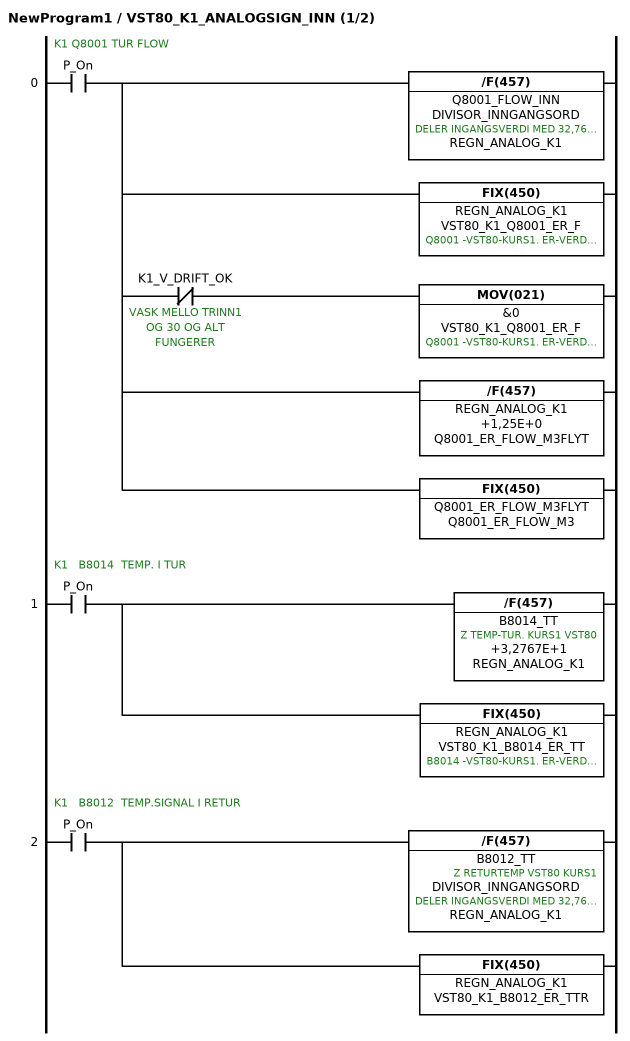
; [picture p144: NewProgram1 / VST80_K1_ANALOGSIGN_INN, rungs 0-2]
; rung 0: K1 Q8001 TUR FLOW
LD P_On
OUT TR0
/F(457) Q8001_FLOW_INN DIVISOR_INNGANGSORD REGN_ANALOG_K1  ; DELER INGANGSVERDI MED 32,760 FOR OMREGNING TIL 0-1000
FIX(450) REGN_ANALOG_K1 VST80_K1_Q8001_ER_F  ; Q8001 -VST80-KURS1. ER-VERDI FLOW I TUR
ANDNOT K1_V_DRIFT_OK  ; VASK MELLO TRINN1 OG 30 OG ALT FUNGERER
MOV(021) &0 VST80_K1_Q8001_ER_F  ; Q8001 -VST80-KURS1. ER-VERDI FLOW I TUR
LD TR0
/F(457) REGN_ANALOG_K1 +1,25E+0 Q8001_ER_FLOW_M3FLYT
FIX(450) Q8001_ER_FLOW_M3FLYT Q8001_ER_FLOW_M3
; rung 1: K1   B8014  TEMP. I TUR
LD P_On
/F(457) B8014_TT +3,2767E+1 REGN_ANALOG_K1  ; Z TEMP-TUR. KURS1 VST80
FIX(450) REGN_ANALOG_K1 VST80_K1_B8014_ER_TT  ; B8014 -VST80-KURS1. ER-VERDI TEMPERATUR I TUR TIL VST
; rung 2: K1   B8012  TEMP.SIGNAL I RETUR
LD P_On
/F(457) B8012_TT DIVISOR_INNGANGSORD REGN_ANALOG_K1  ; Z RETURTEMP VST80 KURS1, DELER INGANGSVERDI MED 32,760 FOR OMREGNING TIL 0-1000
FIX(450) REGN_ANALOG_K1 VST80_K1_B8012_ER_TTR

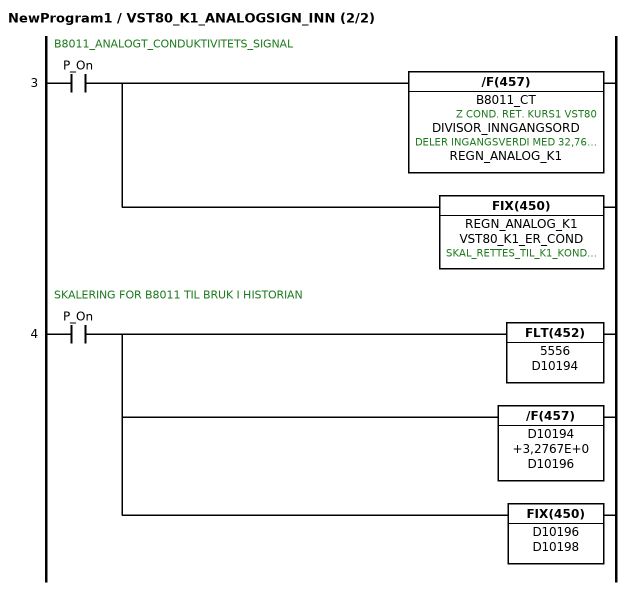
; rung 3: B8011_ANALOGT_CONDUKTIVITETS_SIGNAL
LD P_On
/F(457) B8011_CT DIVISOR_INNGANGSORD REGN_ANALOG_K1  ; Z COND. RET. KURS1 VST80, DELER INGANGSVERDI MED 32,760 FOR OMREGNING TIL 0-1000
FIX(450) REGN_ANALOG_K1 VST80_K1_ER_COND  ; SKAL_RETTES_TIL_K1_KOND_ERVERDI
; rung 4: SKALERING FOR B8011 TIL BRUK I HISTORIAN
LD P_On
FLT(452) 5556 D10194
/F(457) D10194 +3,2767E+0 D10196
FIX(450) D10196 D10198

### Section VST80_K1_GRAF_FEIL_TXT

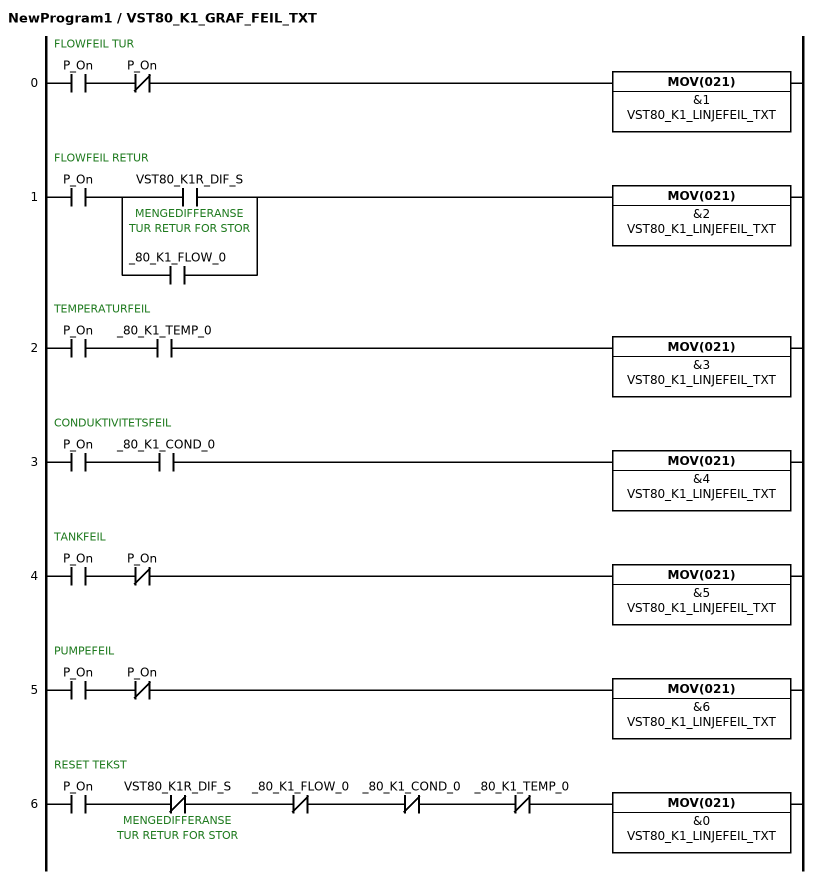
; rung 0: FLOWFEIL TUR
LD P_On
ANDNOT P_On
MOV(021) &1 VST80_K1_LINJEFEIL_TXT
; rung 1: FLOWFEIL RETUR
LD P_On
LD VST80_K1R_DIF_S  ; MENGEDIFFERANSE TUR RETUR FOR STOR
OR _80_K1_FLOW_0
ANDLD
MOV(021) &2 VST80_K1_LINJEFEIL_TXT
; rung 2: TEMPERATURFEIL
LD P_On
AND _80_K1_TEMP_0
MOV(021) &3 VST80_K1_LINJEFEIL_TXT
; rung 3: CONDUKTIVITETSFEIL
LD P_On
AND _80_K1_COND_0
MOV(021) &4 VST80_K1_LINJEFEIL_TXT
; rung 4: TANKFEIL
LD P_On
ANDNOT P_On
MOV(021) &5 VST80_K1_LINJEFEIL_TXT
; rung 5: PUMPEFEIL
LD P_On
ANDNOT P_On
MOV(021) &6 VST80_K1_LINJEFEIL_TXT
; rung 6: RESET TEKST
LD P_On
ANDNOT VST80_K1R_DIF_S  ; MENGEDIFFERANSE TUR RETUR FOR STOR
ANDNOT _80_K1_FLOW_0
ANDNOT _80_K1_COND_0
ANDNOT _80_K1_TEMP_0
MOV(021) &0 VST80_K1_LINJEFEIL_TXT

### Section VST80_K1_MENGDE_FASESKIFT

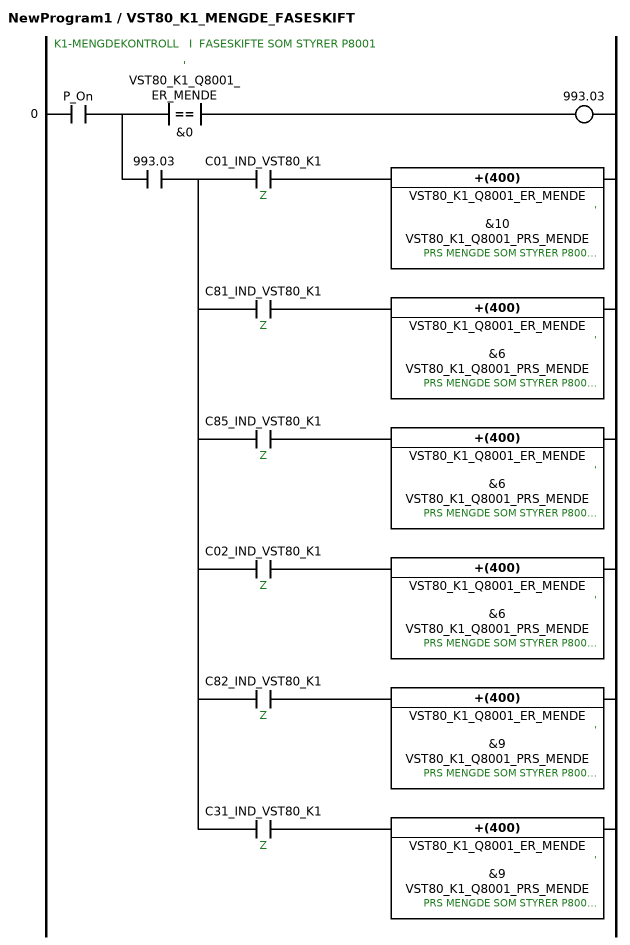
; rung 0: K1-MENGDEKONTROLL   I  FASESKIFTE SOM STYRER P8001
LD P_On
OUT TR0
AND=(300) VST80_K1_Q8001_ER_MENDE &0  ; '
OUT 993.03
LD TR0
AND 993.03
OUT TR0
AND C01_IND_VST80_K1  ; Z
+(400) VST80_K1_Q8001_ER_MENDE &10 VST80_K1_Q8001_PRS_MENDE  ; ', PRS MENGDE SOM STYRER P8001 VED FASESKIFTE
LD TR0
AND C81_IND_VST80_K1  ; Z
+(400) VST80_K1_Q8001_ER_MENDE &6 VST80_K1_Q8001_PRS_MENDE  ; ', PRS MENGDE SOM STYRER P8001 VED FASESKIFTE
LD TR0
AND C85_IND_VST80_K1  ; Z
+(400) VST80_K1_Q8001_ER_MENDE &6 VST80_K1_Q8001_PRS_MENDE  ; ', PRS MENGDE SOM STYRER P8001 VED FASESKIFTE
LD TR0
AND C02_IND_VST80_K1  ; Z
+(400) VST80_K1_Q8001_ER_MENDE &6 VST80_K1_Q8001_PRS_MENDE  ; ', PRS MENGDE SOM STYRER P8001 VED FASESKIFTE
LD TR0
AND C82_IND_VST80_K1  ; Z
+(400) VST80_K1_Q8001_ER_MENDE &9 VST80_K1_Q8001_PRS_MENDE  ; ', PRS MENGDE SOM STYRER P8001 VED FASESKIFTE
LD TR0
AND C31_IND_VST80_K1  ; Z
+(400) VST80_K1_Q8001_ER_MENDE &9 VST80_K1_Q8001_PRS_MENDE  ; ', PRS MENGDE SOM STYRER P8001 VED FASESKIFTE

### Section VST80_K1_TR_VEKS
; VST80 KURS1 VEKSLING AV TRINN.

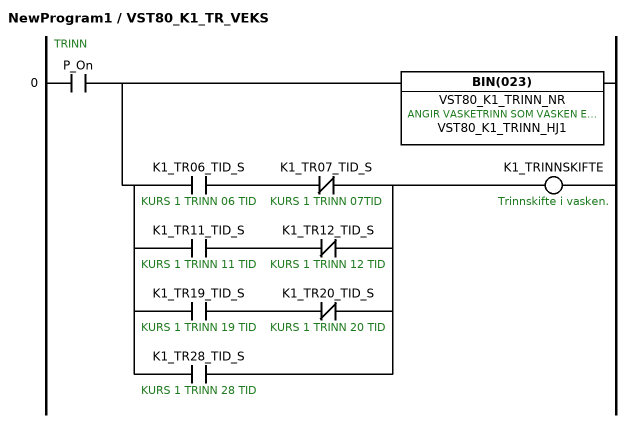
; rung 0: TRINN
LD P_On
BIN(023) VST80_K1_TRINN_NR VST80_K1_TRINN_HJ1  ; ANGIR VASKETRINN SOM VASKEN ER I
LD K1_TR06_TID_S  ; KURS 1 TRINN 06 TID
ANDNOT K1_TR07_TID_S  ; KURS 1 TRINN 07TID
LD K1_TR11_TID_S  ; KURS 1 TRINN 11 TID
ANDNOT K1_TR12_TID_S  ; KURS 1 TRINN 12 TID
ORLD
LD K1_TR19_TID_S  ; KURS 1 TRINN 19 TID
ANDNOT K1_TR20_TID_S  ; KURS 1 TRINN 20 TID
ORLD
OR K1_TR28_TID_S  ; KURS 1 TRINN 28 TID
ANDLD
OUT K1_TRINNSKIFTE  ; Trinnskifte i vasken.

### Section VST80_K1_FEIL_RET
; FEIL I RETUR / FLOW / TEMP / COND

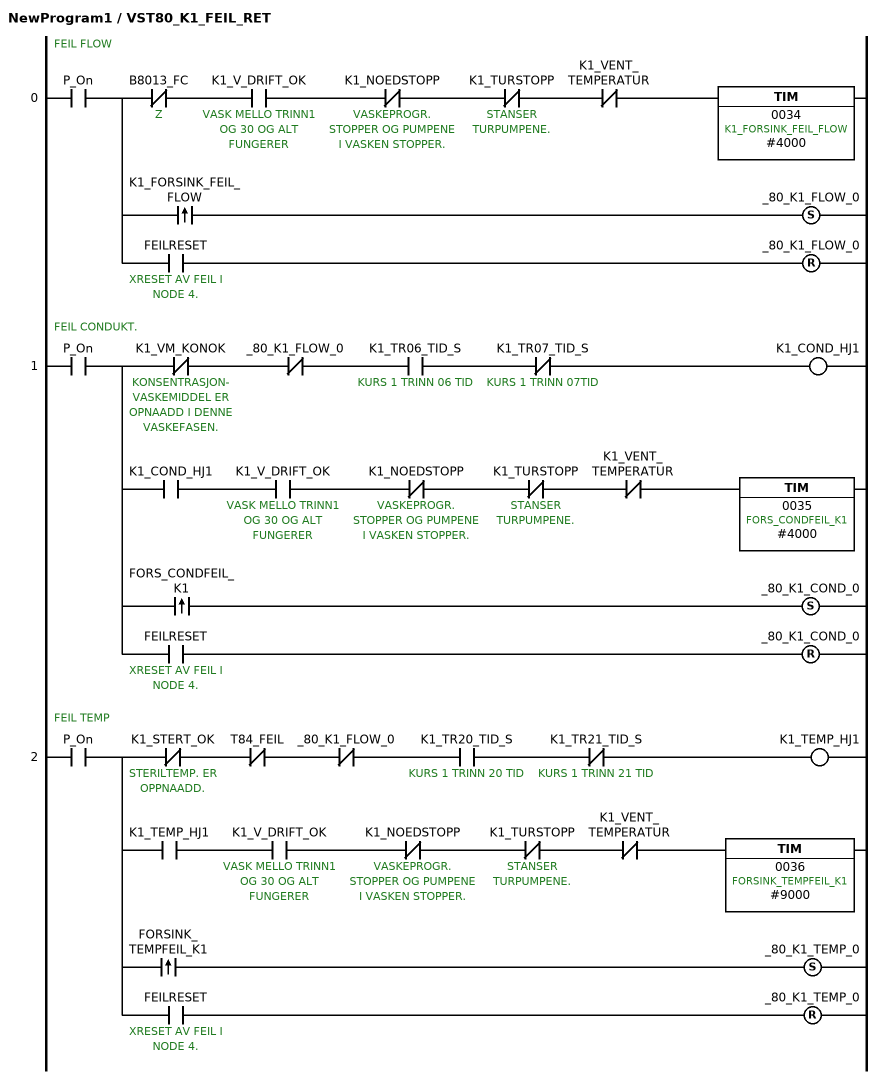
; rung 0: FEIL FLOW
LD P_On
OUT TR0
ANDNOT B8013_FC  ; Z
AND K1_V_DRIFT_OK  ; VASK MELLO TRINN1 OG 30 OG ALT FUNGERER
ANDNOT K1_NOEDSTOPP  ; VASKEPROGR. STOPPER OG PUMPENE I VASKEN STOPPER.
ANDNOT K1_TURSTOPP  ; STANSER TURPUMPENE.
ANDNOT K1_VENT_TEMPERATUR
TIM 0034 #4000  ; K1_FORSINK_FEIL_FLOW
LD TR0
@AND K1_FORSINK_FEIL_FLOW
SET _80_K1_FLOW_0
LD TR0
AND FEILRESET  ; XRESET AV FEIL I NODE 4.
RSET _80_K1_FLOW_0
; rung 1: FEIL CONDUKT.
LD P_On
OUT TR0
ANDNOT K1_VM_KONOK  ; KONSENTRASJON-VASKEMIDDEL ER OPNAADD I DENNE VASKEFASEN.
ANDNOT _80_K1_FLOW_0
AND K1_TR06_TID_S  ; KURS 1 TRINN 06 TID
ANDNOT K1_TR07_TID_S  ; KURS 1 TRINN 07TID
OUT K1_COND_HJ1
LD TR0
AND K1_COND_HJ1
AND K1_V_DRIFT_OK  ; VASK MELLO TRINN1 OG 30 OG ALT FUNGERER
ANDNOT K1_NOEDSTOPP  ; VASKEPROGR. STOPPER OG PUMPENE I VASKEN STOPPER.
ANDNOT K1_TURSTOPP  ; STANSER TURPUMPENE.
ANDNOT K1_VENT_TEMPERATUR
TIM 0035 #4000  ; FORS_CONDFEIL_K1
LD TR0
@AND FORS_CONDFEIL_K1
SET _80_K1_COND_0
LD TR0
AND FEILRESET  ; XRESET AV FEIL I NODE 4.
RSET _80_K1_COND_0
; rung 2: FEIL TEMP
LD P_On
OUT TR0
ANDNOT K1_STERT_OK  ; STERILTEMP. ER OPPNAADD.
ANDNOT T84_FEIL
ANDNOT _80_K1_FLOW_0
AND K1_TR20_TID_S  ; KURS 1 TRINN 20 TID
ANDNOT K1_TR21_TID_S  ; KURS 1 TRINN 21 TID
OUT K1_TEMP_HJ1
LD TR0
AND K1_TEMP_HJ1
AND K1_V_DRIFT_OK  ; VASK MELLO TRINN1 OG 30 OG ALT FUNGERER
ANDNOT K1_NOEDSTOPP  ; VASKEPROGR. STOPPER OG PUMPENE I VASKEN STOPPER.
ANDNOT K1_TURSTOPP  ; STANSER TURPUMPENE.
ANDNOT K1_VENT_TEMPERATUR
TIM 0036 #9000  ; FORSINK_TEMPFEIL_K1
LD TR0
@AND FORSINK_TEMPFEIL_K1
SET _80_K1_TEMP_0
LD TR0
AND FEILRESET  ; XRESET AV FEIL I NODE 4.
RSET _80_K1_TEMP_0

### Section VST80_K1_VASKERAPPORT
; VST80 / KURS1 VASKERAPPORT

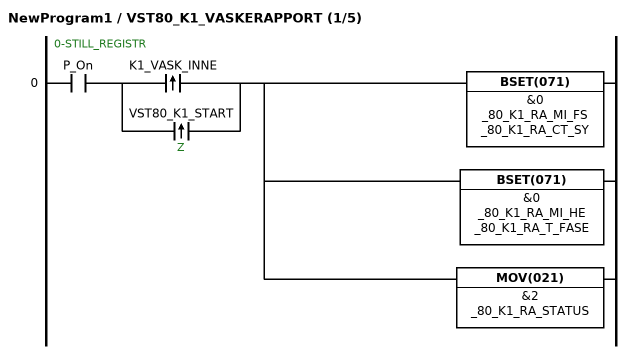
; rung 0: 0-STILL_REGISTR
LD P_On
@LD K1_VASK_INNE
@OR VST80_K1_START  ; Z
ANDLD
BSET(071) &0 _80_K1_RA_MI_FS _80_K1_RA_CT_SY
BSET(071) &0 _80_K1_RA_MI_HE _80_K1_RA_T_FASE
MOV(021) &2 _80_K1_RA_STATUS

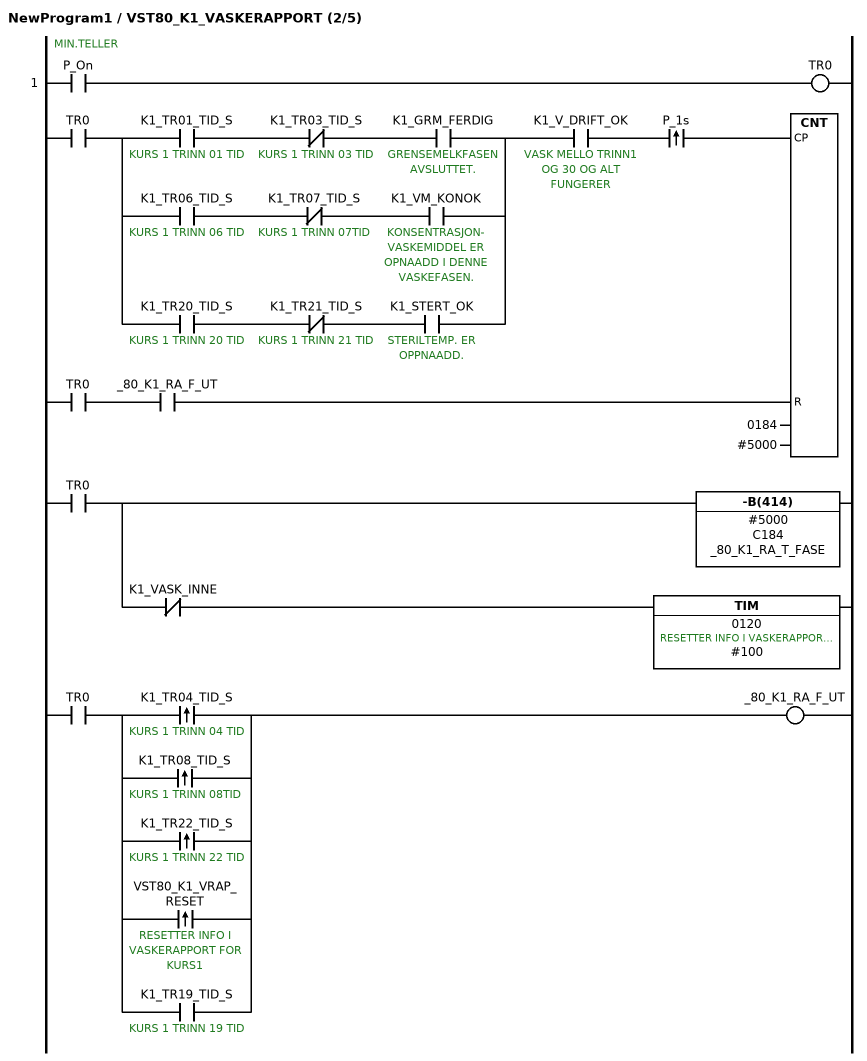
; rung 1: MIN.TELLER
LD P_On
OUT TR0
LD K1_TR01_TID_S  ; KURS 1 TRINN 01 TID
ANDNOT K1_TR03_TID_S  ; KURS 1 TRINN 03 TID
AND K1_GRM_FERDIG  ; GRENSEMELKFASEN AVSLUTTET.
LD K1_TR06_TID_S  ; KURS 1 TRINN 06 TID
ANDNOT K1_TR07_TID_S  ; KURS 1 TRINN 07TID
AND K1_VM_KONOK  ; KONSENTRASJON-VASKEMIDDEL ER OPNAADD I DENNE VASKEFASEN.
ORLD
LD K1_TR20_TID_S  ; KURS 1 TRINN 20 TID
ANDNOT K1_TR21_TID_S  ; KURS 1 TRINN 21 TID
AND K1_STERT_OK  ; STERILTEMP. ER OPPNAADD.
ORLD
ANDLD
AND K1_V_DRIFT_OK  ; VASK MELLO TRINN1 OG 30 OG ALT FUNGERER
@AND P_1s
LD TR0
AND _80_K1_RA_F_UT
CNT 0184 #5000
LD TR0
-B(414) #5000 C184 _80_K1_RA_T_FASE
ANDNOT K1_VASK_INNE
TIM 0120 #100  ; RESETTER INFO I VASKERAPPORT FOR KURS1
LD TR0
@LD K1_TR04_TID_S  ; KURS 1 TRINN 04 TID
@OR K1_TR08_TID_S  ; KURS 1 TRINN 08TID
@OR K1_TR22_TID_S  ; KURS 1 TRINN 22 TID
@OR VST80_K1_VRAP_RESET  ; RESETTER INFO I VASKERAPPORT FOR KURS1
OR K1_TR19_TID_S  ; KURS 1 TRINN 19 TID
ANDLD
OUT _80_K1_RA_F_UT

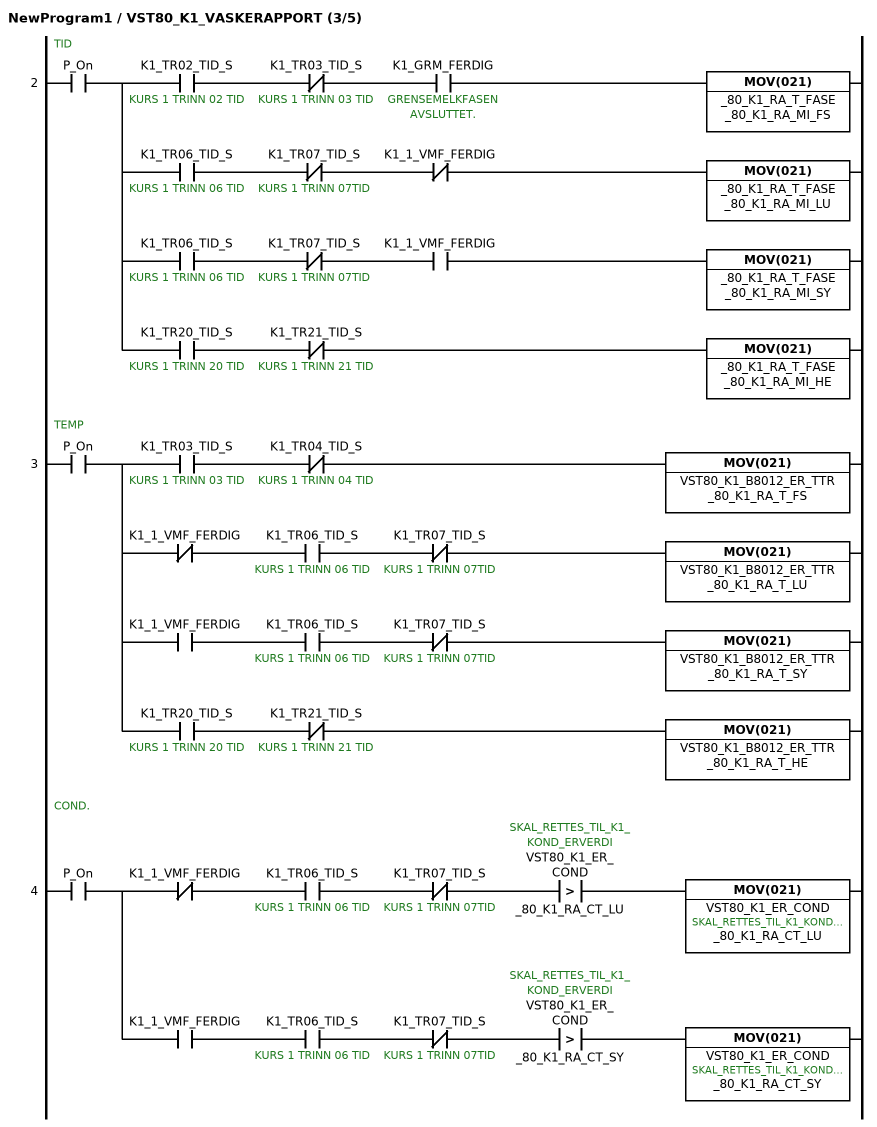
; rung 2: TID
LD P_On
OUT TR0
AND K1_TR02_TID_S  ; KURS 1 TRINN 02 TID
ANDNOT K1_TR03_TID_S  ; KURS 1 TRINN 03 TID
AND K1_GRM_FERDIG  ; GRENSEMELKFASEN AVSLUTTET.
MOV(021) _80_K1_RA_T_FASE _80_K1_RA_MI_FS
LD TR0
AND K1_TR06_TID_S  ; KURS 1 TRINN 06 TID
ANDNOT K1_TR07_TID_S  ; KURS 1 TRINN 07TID
ANDNOT K1_1_VMF_FERDIG
MOV(021) _80_K1_RA_T_FASE _80_K1_RA_MI_LU
LD TR0
AND K1_TR06_TID_S  ; KURS 1 TRINN 06 TID
ANDNOT K1_TR07_TID_S  ; KURS 1 TRINN 07TID
AND K1_1_VMF_FERDIG
MOV(021) _80_K1_RA_T_FASE _80_K1_RA_MI_SY
LD TR0
AND K1_TR20_TID_S  ; KURS 1 TRINN 20 TID
ANDNOT K1_TR21_TID_S  ; KURS 1 TRINN 21 TID
MOV(021) _80_K1_RA_T_FASE _80_K1_RA_MI_HE
; rung 3: TEMP
LD P_On
OUT TR0
AND K1_TR03_TID_S  ; KURS 1 TRINN 03 TID
ANDNOT K1_TR04_TID_S  ; KURS 1 TRINN 04 TID
MOV(021) VST80_K1_B8012_ER_TTR _80_K1_RA_T_FS
LD TR0
ANDNOT K1_1_VMF_FERDIG
AND K1_TR06_TID_S  ; KURS 1 TRINN 06 TID
ANDNOT K1_TR07_TID_S  ; KURS 1 TRINN 07TID
MOV(021) VST80_K1_B8012_ER_TTR _80_K1_RA_T_LU
LD TR0
AND K1_1_VMF_FERDIG
AND K1_TR06_TID_S  ; KURS 1 TRINN 06 TID
ANDNOT K1_TR07_TID_S  ; KURS 1 TRINN 07TID
MOV(021) VST80_K1_B8012_ER_TTR _80_K1_RA_T_SY
LD TR0
AND K1_TR20_TID_S  ; KURS 1 TRINN 20 TID
ANDNOT K1_TR21_TID_S  ; KURS 1 TRINN 21 TID
MOV(021) VST80_K1_B8012_ER_TTR _80_K1_RA_T_HE
; rung 4: COND.
LD P_On
OUT TR0
ANDNOT K1_1_VMF_FERDIG
AND K1_TR06_TID_S  ; KURS 1 TRINN 06 TID
ANDNOT K1_TR07_TID_S  ; KURS 1 TRINN 07TID
AND>(320) VST80_K1_ER_COND _80_K1_RA_CT_LU  ; SKAL_RETTES_TIL_K1_KOND_ERVERDI
MOV(021) VST80_K1_ER_COND _80_K1_RA_CT_LU  ; SKAL_RETTES_TIL_K1_KOND_ERVERDI
LD TR0
AND K1_1_VMF_FERDIG
AND K1_TR06_TID_S  ; KURS 1 TRINN 06 TID
ANDNOT K1_TR07_TID_S  ; KURS 1 TRINN 07TID
AND>(320) VST80_K1_ER_COND _80_K1_RA_CT_SY  ; SKAL_RETTES_TIL_K1_KOND_ERVERDI
MOV(021) VST80_K1_ER_COND _80_K1_RA_CT_SY  ; SKAL_RETTES_TIL_K1_KOND_ERVERDI

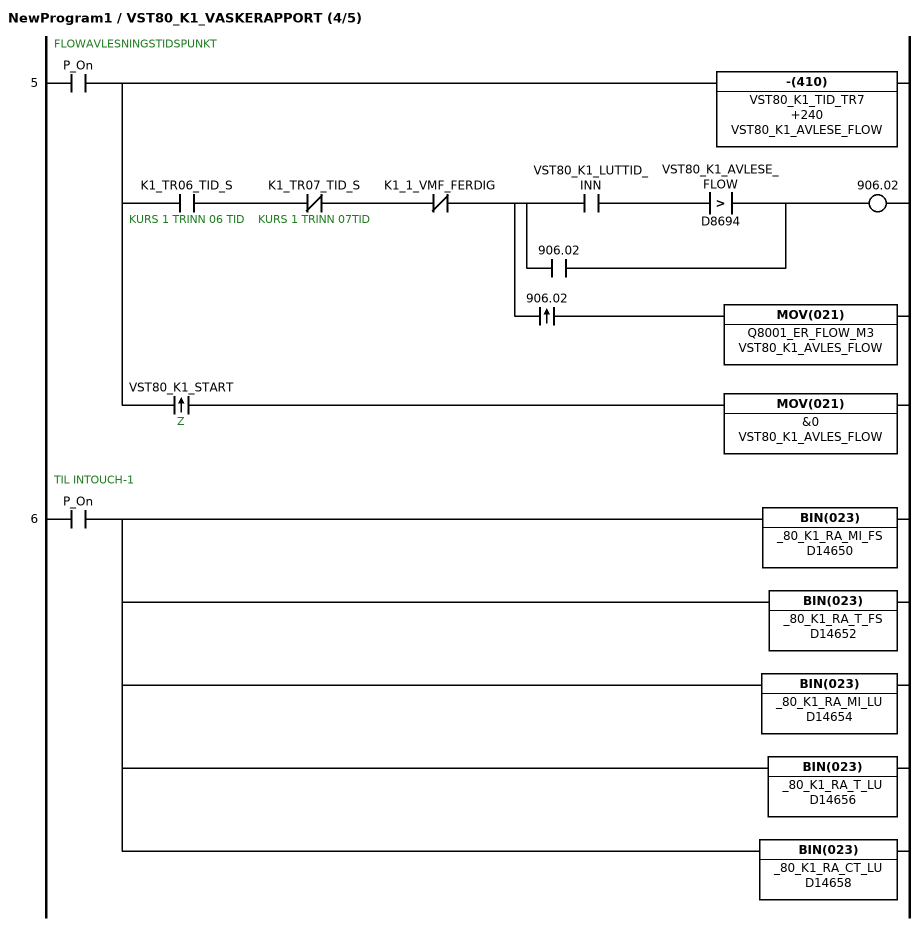
; rung 5: FLOWAVLESNINGSTIDSPUNKT
LD P_On
OUT TR0
-(410) VST80_K1_TID_TR7 +240 VST80_K1_AVLESE_FLOW
AND K1_TR06_TID_S  ; KURS 1 TRINN 06 TID
ANDNOT K1_TR07_TID_S  ; KURS 1 TRINN 07TID
ANDNOT K1_1_VMF_FERDIG
OUT TR1
LD VST80_K1_LUTTID_INN
AND>(320) VST80_K1_AVLESE_FLOW D8694
OR 906.02
ANDLD
OUT 906.02
LD TR1
@AND 906.02
MOV(021) Q8001_ER_FLOW_M3 VST80_K1_AVLES_FLOW
LD TR0
@AND VST80_K1_START  ; Z
MOV(021) &0 VST80_K1_AVLES_FLOW
; rung 6: TIL INTOUCH-1
LD P_On
BIN(023) _80_K1_RA_MI_FS D14650
BIN(023) _80_K1_RA_T_FS D14652
BIN(023) _80_K1_RA_MI_LU D14654
BIN(023) _80_K1_RA_T_LU D14656
BIN(023) _80_K1_RA_CT_LU D14658

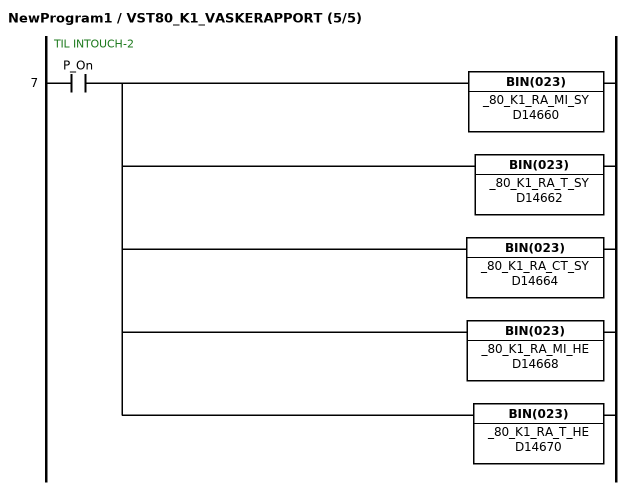
; rung 7: TIL INTOUCH-2
LD P_On
BIN(023) _80_K1_RA_MI_SY D14660
BIN(023) _80_K1_RA_T_SY D14662
BIN(023) _80_K1_RA_CT_SY D14664
BIN(023) _80_K1_RA_MI_HE D14668
BIN(023) _80_K1_RA_T_HE D14670

### Section VST80_K1_REGULATORER

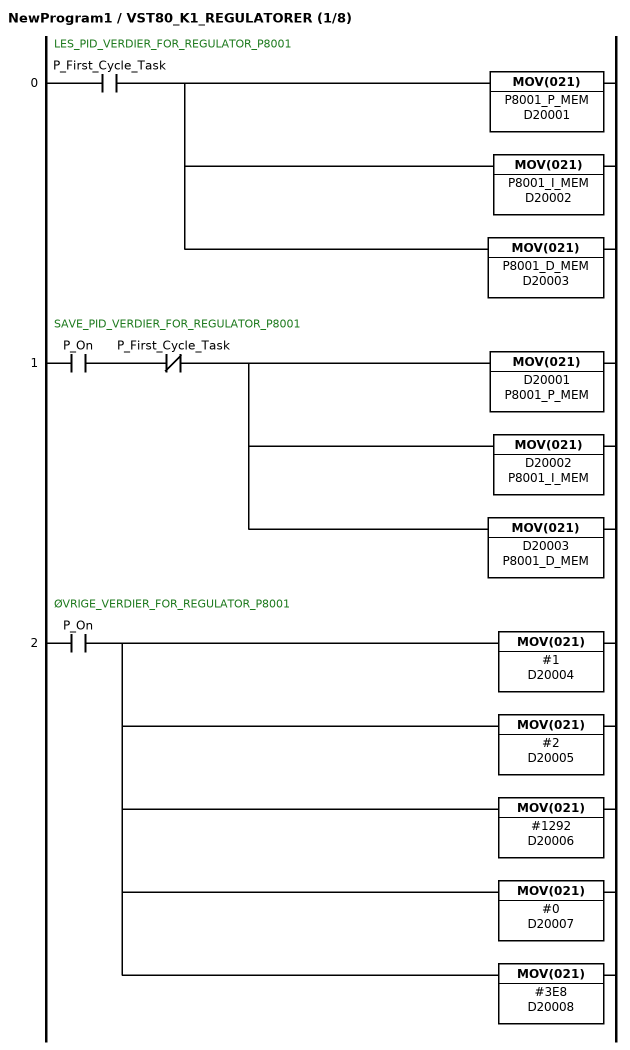
; rung 0: LES_PID_VERDIER_FOR_REGULATOR_P8001
LD P_First_Cycle_Task
MOV(021) P8001_P_MEM D20001
MOV(021) P8001_I_MEM D20002
MOV(021) P8001_D_MEM D20003
; rung 1: SAVE_PID_VERDIER_FOR_REGULATOR_P8001
LD P_On
ANDNOT P_First_Cycle_Task
MOV(021) D20001 P8001_P_MEM
MOV(021) D20002 P8001_I_MEM
MOV(021) D20003 P8001_D_MEM
; rung 2: ØVRIGE_VERDIER_FOR_REGULATOR_P8001
LD P_On
MOV(021) #1 D20004
MOV(021) #2 D20005
MOV(021) #1292 D20006
MOV(021) #0 D20007
MOV(021) #3E8 D20008

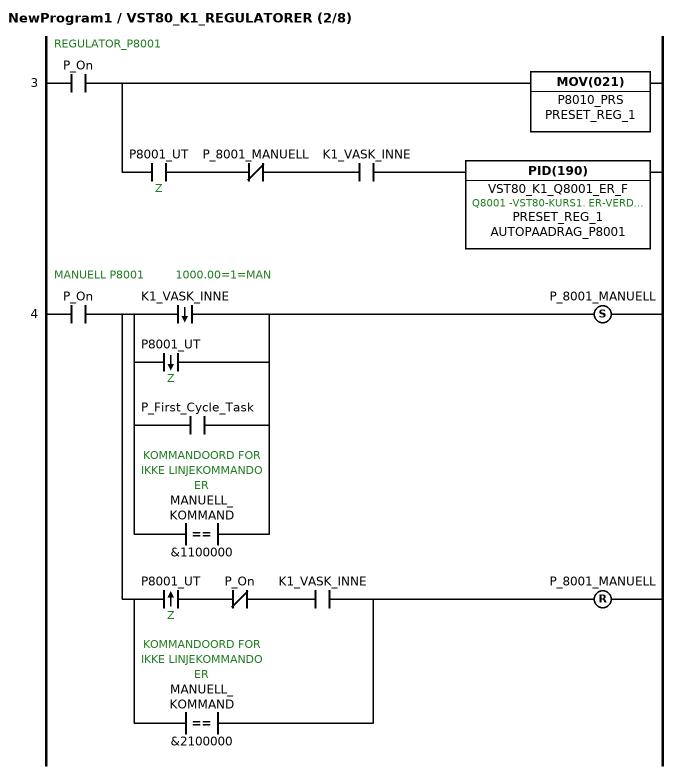
; rung 3: REGULATOR_P8001
LD P_On
MOV(021) P8010_PRS PRESET_REG_1
AND P8001_UT  ; Z
ANDNOT P_8001_MANUELL
AND K1_VASK_INNE
PID(190) VST80_K1_Q8001_ER_F PRESET_REG_1 AUTOPAADRAG_P8001  ; Q8001 -VST80-KURS1. ER-VERDI FLOW I TUR
; rung 4: MANUELL P8001         1000.00=1=MAN
LD P_On
OUT TR0
%LD K1_VASK_INNE
%OR P8001_UT  ; Z
OR P_First_Cycle_Task
OR=L(301) MANUELL_KOMMAND &1100000  ; KOMMANDOORD FOR IKKE LINJEKOMMANDOER
ANDLD
SET P_8001_MANUELL
LD TR0
@LD P8001_UT  ; Z
ANDNOT P_On
AND K1_VASK_INNE
OR=L(301) MANUELL_KOMMAND &2100000  ; KOMMANDOORD FOR IKKE LINJEKOMMANDOER
ANDLD
RSET P_8001_MANUELL

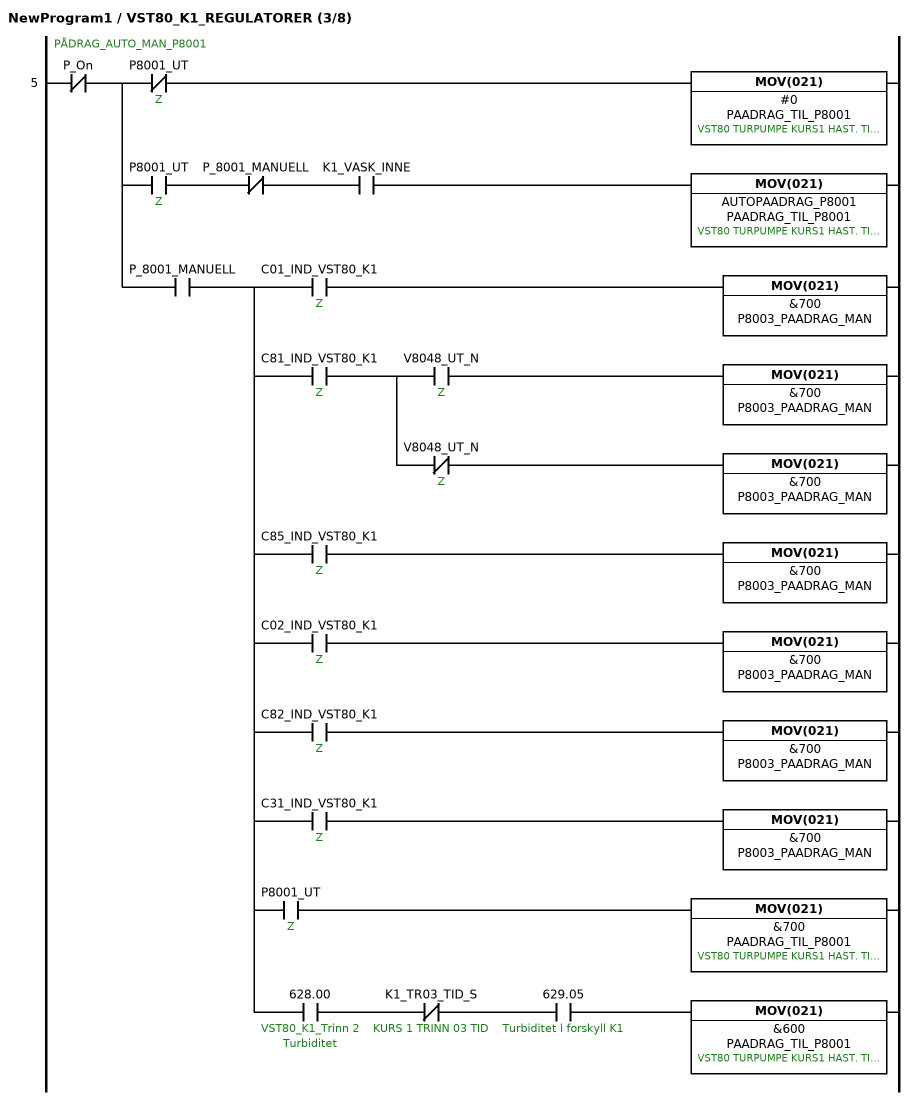
; rung 5: PÅDRAG_AUTO_MAN_P8001
LDNOT P_On
OUT TR0
ANDNOT P8001_UT  ; Z
MOV(021) #0 PAADRAG_TIL_P8001  ; VST80 TURPUMPE KURS1 HAST. TIL FR.OMF. P8010
LD TR0
AND P8001_UT  ; Z
ANDNOT P_8001_MANUELL
AND K1_VASK_INNE
MOV(021) AUTOPAADRAG_P8001 PAADRAG_TIL_P8001  ; VST80 TURPUMPE KURS1 HAST. TIL FR.OMF. P8010
LD TR0
AND P_8001_MANUELL
OUT TR0
AND C01_IND_VST80_K1  ; Z
MOV(021) &700 P8003_PAADRAG_MAN
LD TR0
AND C81_IND_VST80_K1  ; Z
OUT TR1
AND V8048_UT_N  ; Z
MOV(021) &700 P8003_PAADRAG_MAN
LD TR1
ANDNOT V8048_UT_N  ; Z
MOV(021) &700 P8003_PAADRAG_MAN
LD TR0
AND C85_IND_VST80_K1  ; Z
MOV(021) &700 P8003_PAADRAG_MAN
LD TR0
AND C02_IND_VST80_K1  ; Z
MOV(021) &700 P8003_PAADRAG_MAN
LD TR0
AND C82_IND_VST80_K1  ; Z
MOV(021) &700 P8003_PAADRAG_MAN
LD TR0
AND C31_IND_VST80_K1  ; Z
MOV(021) &700 P8003_PAADRAG_MAN
LD TR0
AND P8001_UT  ; Z
MOV(021) &700 PAADRAG_TIL_P8001  ; VST80 TURPUMPE KURS1 HAST. TIL FR.OMF. P8010
LD TR0
AND 628.00  ; VST80_K1_Trinn 2 Turbiditet
ANDNOT K1_TR03_TID_S  ; KURS 1 TRINN 03 TID
AND 629.05  ; Turbiditet i forskyll K1
MOV(021) &600 PAADRAG_TIL_P8001  ; VST80 TURPUMPE KURS1 HAST. TIL FR.OMF. P8010

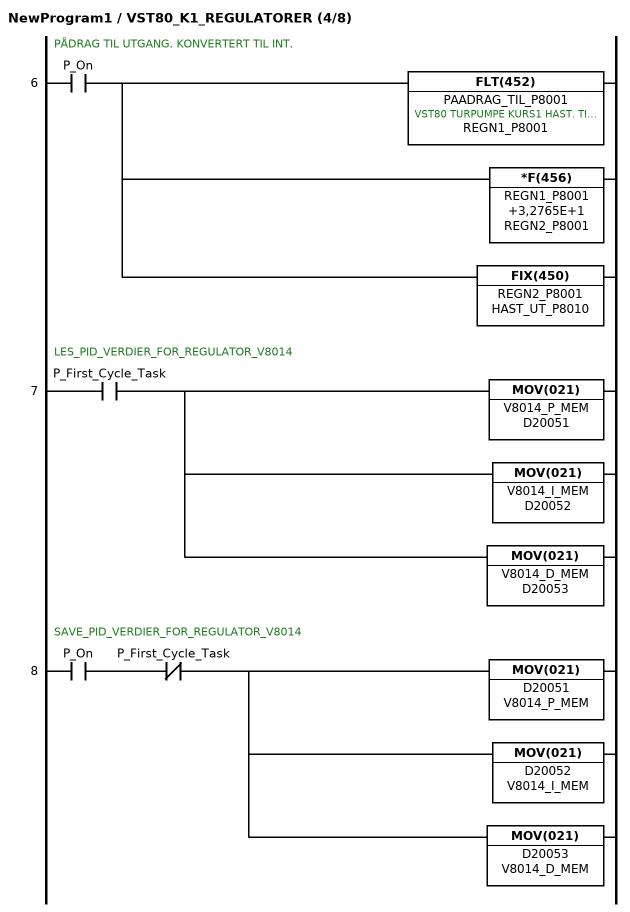
; rung 6: PÅDRAG TIL UTGANG. KONVERTERT TIL INT.
LD P_On
FLT(452) PAADRAG_TIL_P8001 REGN1_P8001  ; VST80 TURPUMPE KURS1 HAST. TIL FR.OMF. P8010
*F(456) REGN1_P8001 +3,2765E+1 REGN2_P8001
FIX(450) REGN2_P8001 HAST_UT_P8010
; rung 7: LES_PID_VERDIER_FOR_REGULATOR_V8014
LD P_First_Cycle_Task
MOV(021) V8014_P_MEM D20051
MOV(021) V8014_I_MEM D20052
MOV(021) V8014_D_MEM D20053
; rung 8: SAVE_PID_VERDIER_FOR_REGULATOR_V8014
LD P_On
ANDNOT P_First_Cycle_Task
MOV(021) D20051 V8014_P_MEM
MOV(021) D20052 V8014_I_MEM
MOV(021) D20053 V8014_D_MEM

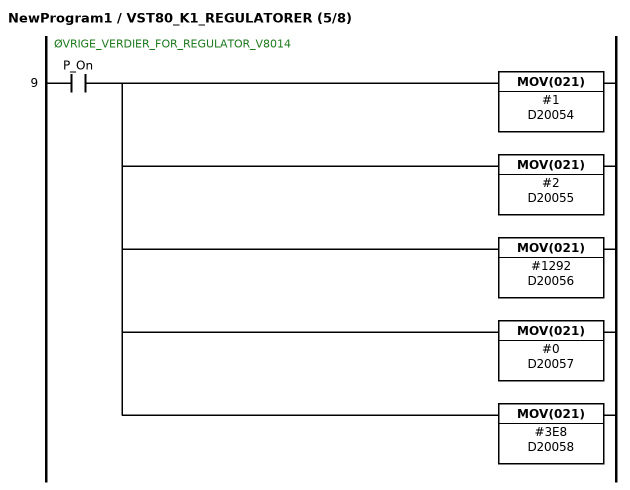
; rung 9: ØVRIGE_VERDIER_FOR_REGULATOR_V8014
LD P_On
MOV(021) #1 D20054
MOV(021) #2 D20055
MOV(021) #1292 D20056
MOV(021) #0 D20057
MOV(021) #3E8 D20058

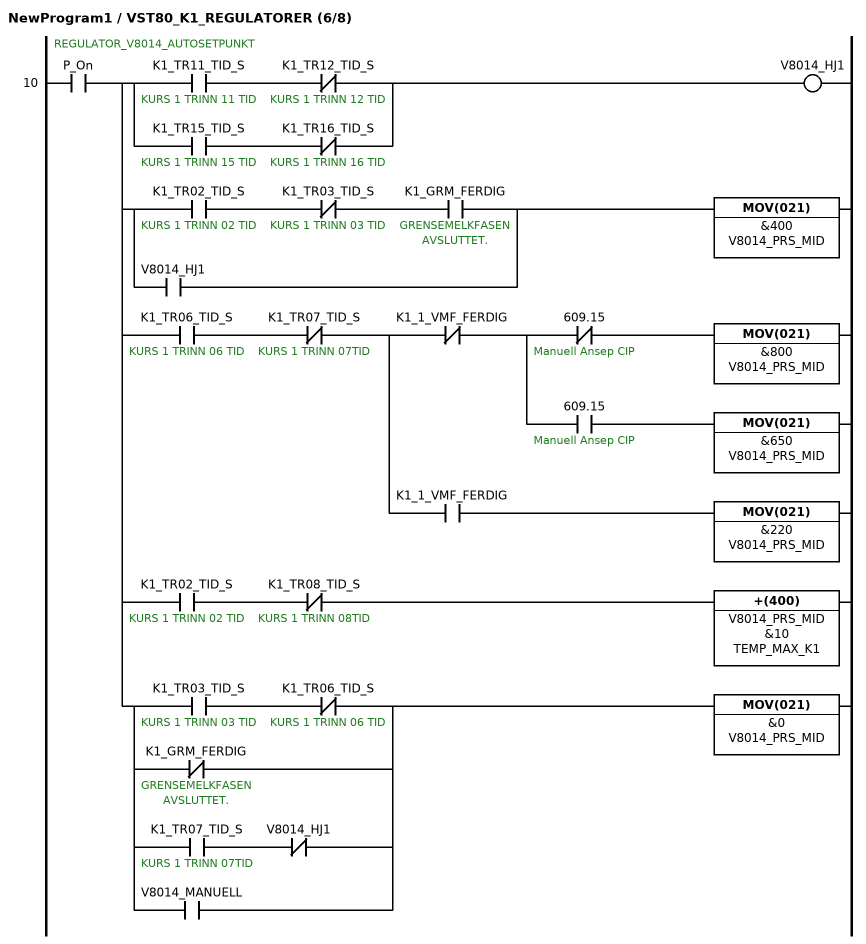
; rung 10: REGULATOR_V8014_AUTOSETPUNKT
LD P_On
OUT TR0
LD K1_TR11_TID_S  ; KURS 1 TRINN 11 TID
ANDNOT K1_TR12_TID_S  ; KURS 1 TRINN 12 TID
LD K1_TR15_TID_S  ; KURS 1 TRINN 15 TID
ANDNOT K1_TR16_TID_S  ; KURS 1 TRINN 16 TID
ORLD
ANDLD
OUT V8014_HJ1
LD TR0
LD K1_TR02_TID_S  ; KURS 1 TRINN 02 TID
ANDNOT K1_TR03_TID_S  ; KURS 1 TRINN 03 TID
AND K1_GRM_FERDIG  ; GRENSEMELKFASEN AVSLUTTET.
OR V8014_HJ1
ANDLD
MOV(021) &400 V8014_PRS_MID
LD TR0
AND K1_TR06_TID_S  ; KURS 1 TRINN 06 TID
ANDNOT K1_TR07_TID_S  ; KURS 1 TRINN 07TID
OUT TR1
ANDNOT K1_1_VMF_FERDIG
OUT TR2
ANDNOT 609.15  ; Manuell Ansep CIP
MOV(021) &800 V8014_PRS_MID
LD TR2
AND 609.15  ; Manuell Ansep CIP
MOV(021) &650 V8014_PRS_MID
LD TR1
AND K1_1_VMF_FERDIG
MOV(021) &220 V8014_PRS_MID
LD TR0
AND K1_TR02_TID_S  ; KURS 1 TRINN 02 TID
ANDNOT K1_TR08_TID_S  ; KURS 1 TRINN 08TID
+(400) V8014_PRS_MID &10 TEMP_MAX_K1
LD TR0
LD K1_TR03_TID_S  ; KURS 1 TRINN 03 TID
ANDNOT K1_TR06_TID_S  ; KURS 1 TRINN 06 TID
ORNOT K1_GRM_FERDIG  ; GRENSEMELKFASEN AVSLUTTET.
LD K1_TR07_TID_S  ; KURS 1 TRINN 07TID
ANDNOT V8014_HJ1
ORLD
OR V8014_MANUELL
ANDLD
MOV(021) &0 V8014_PRS_MID

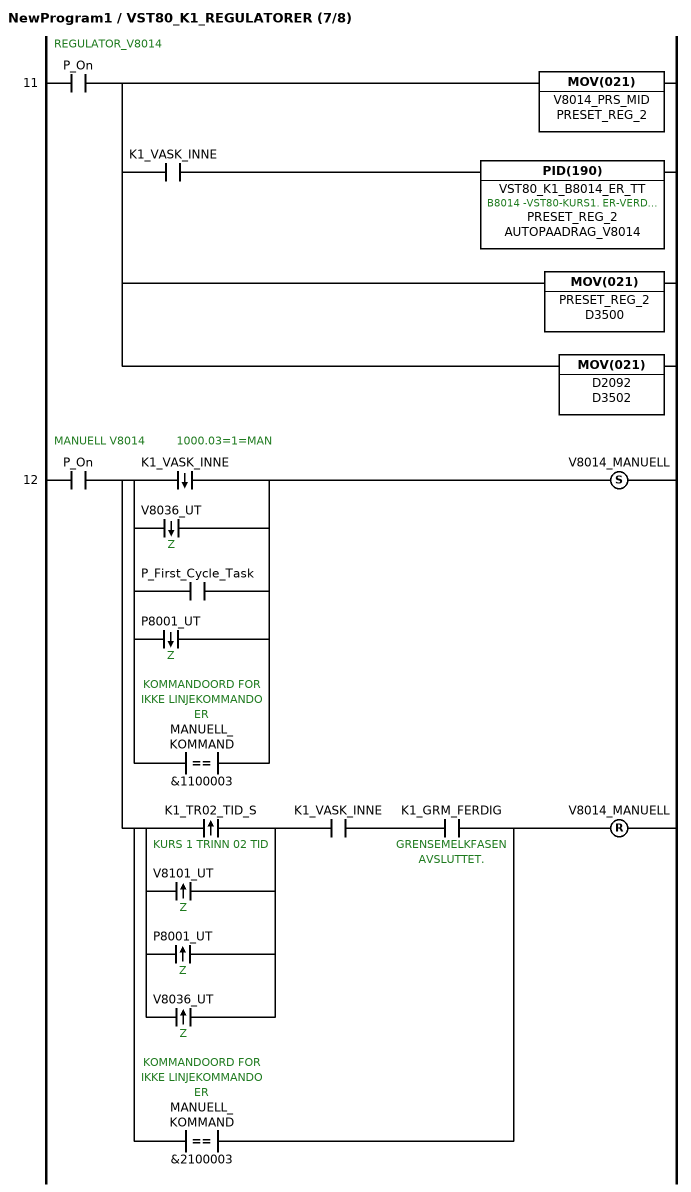
; rung 11: REGULATOR_V8014
LD P_On
OUT TR0
MOV(021) V8014_PRS_MID PRESET_REG_2
AND K1_VASK_INNE
PID(190) VST80_K1_B8014_ER_TT PRESET_REG_2 AUTOPAADRAG_V8014  ; B8014 -VST80-KURS1. ER-VERDI TEMPERATUR I TUR TIL VST
LD TR0
MOV(021) PRESET_REG_2 D3500
MOV(021) D2092 D3502
; rung 12: MANUELL V8014         1000.03=1=MAN
LD P_On
OUT TR0
%LD K1_VASK_INNE
%OR V8036_UT  ; Z
OR P_First_Cycle_Task
%OR P8001_UT  ; Z
OR=L(301) MANUELL_KOMMAND &1100003  ; KOMMANDOORD FOR IKKE LINJEKOMMANDOER
ANDLD
SET V8014_MANUELL
LD TR0
@LD K1_TR02_TID_S  ; KURS 1 TRINN 02 TID
@OR V8101_UT  ; Z
@OR P8001_UT  ; Z
@OR V8036_UT  ; Z
AND K1_VASK_INNE
AND K1_GRM_FERDIG  ; GRENSEMELKFASEN AVSLUTTET.
OR=L(301) MANUELL_KOMMAND &2100003  ; KOMMANDOORD FOR IKKE LINJEKOMMANDOER
ANDLD
RSET V8014_MANUELL

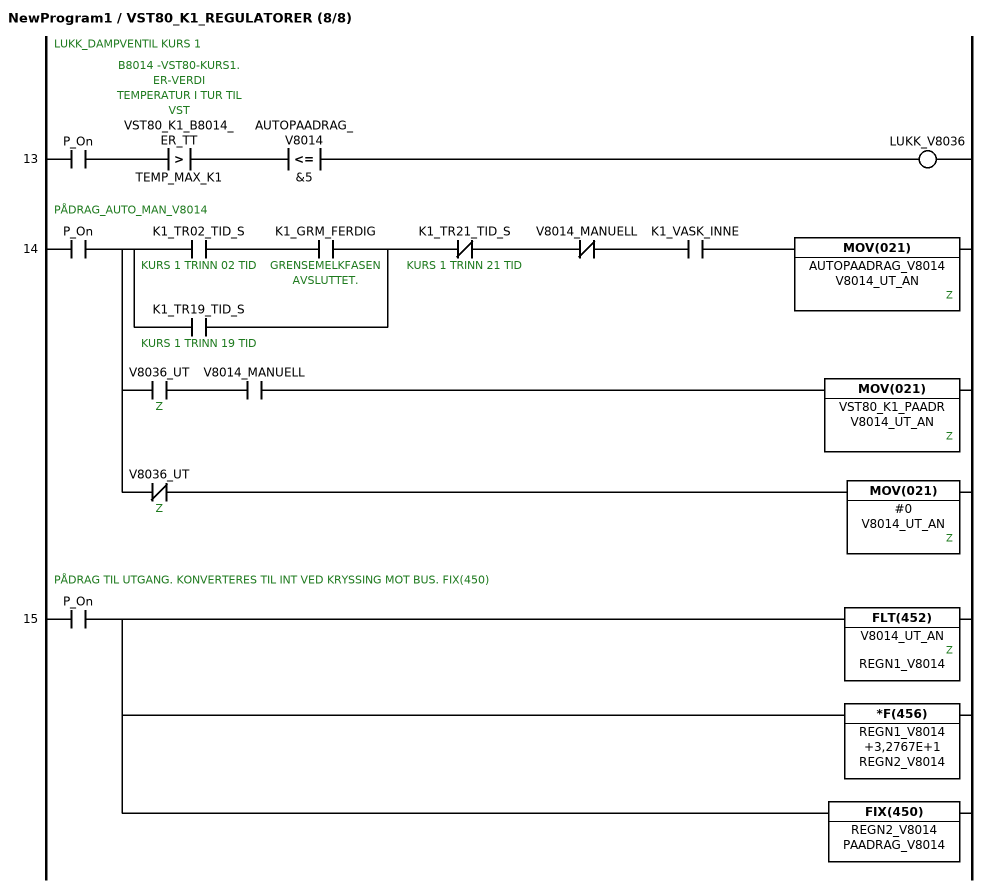
; rung 13: LUKK_DAMPVENTIL KURS 1
LD P_On
AND>(320) VST80_K1_B8014_ER_TT TEMP_MAX_K1  ; B8014 -VST80-KURS1. ER-VERDI TEMPERATUR I TUR TIL VST
AND<=(315) AUTOPAADRAG_V8014 &5
OUT LUKK_V8036
; rung 14: PÅDRAG_AUTO_MAN_V8014
LD P_On
OUT TR0
LD K1_TR02_TID_S  ; KURS 1 TRINN 02 TID
AND K1_GRM_FERDIG  ; GRENSEMELKFASEN AVSLUTTET.
OR K1_TR19_TID_S  ; KURS 1 TRINN 19 TID
ANDLD
ANDNOT K1_TR21_TID_S  ; KURS 1 TRINN 21 TID
ANDNOT V8014_MANUELL
AND K1_VASK_INNE
MOV(021) AUTOPAADRAG_V8014 V8014_UT_AN  ; Z
LD TR0
AND V8036_UT  ; Z
AND V8014_MANUELL
MOV(021) VST80_K1_PAADR V8014_UT_AN  ; Z
LD TR0
ANDNOT V8036_UT  ; Z
MOV(021) #0 V8014_UT_AN  ; Z
; rung 15: PÅDRAG TIL UTGANG. KONVERTERES TIL INT VED KRYSSING MOT BUS. FIX(450)
LD P_On
FLT(452) V8014_UT_AN REGN1_V8014  ; Z
*F(456) REGN1_V8014 +3,2767E+1 REGN2_V8014
FIX(450) REGN2_V8014 PAADRAG_V8014

### Section VST80_K_2_TIDER_TR1_18

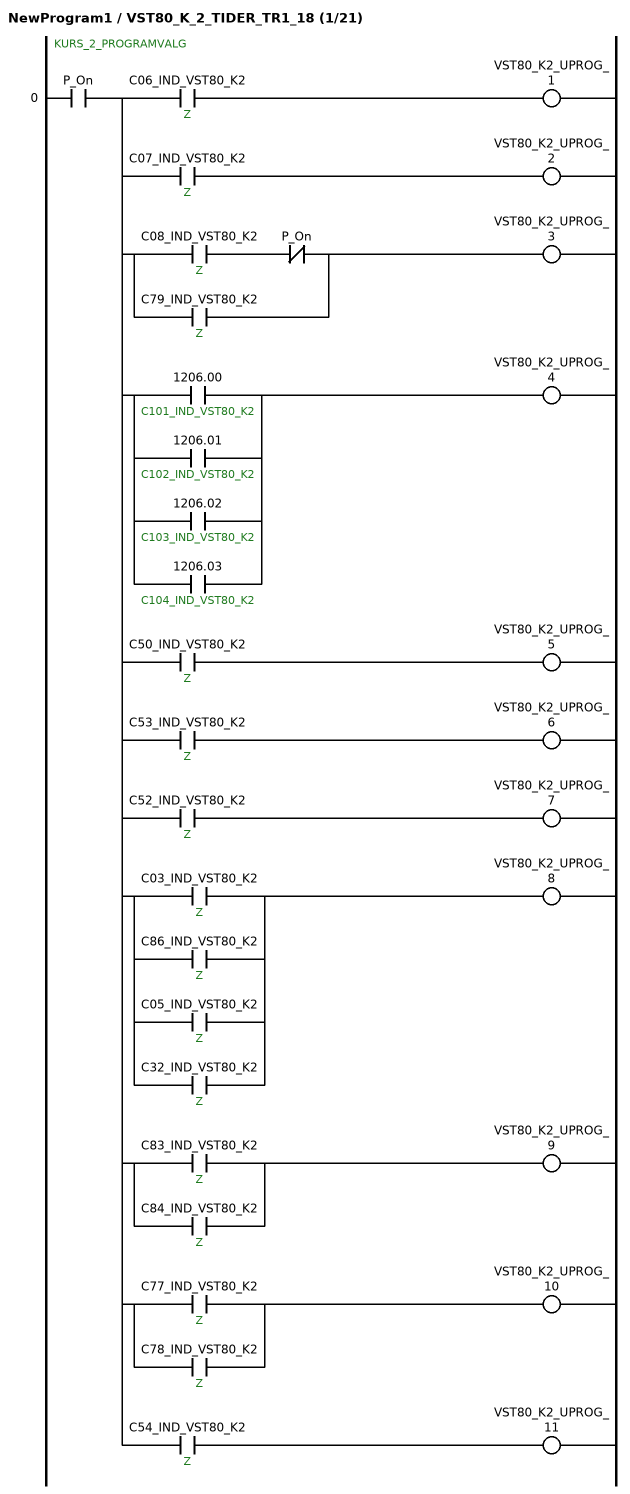
; rung 0: KURS_2_PROGRAMVALG
LD P_On
OUT TR0
AND C06_IND_VST80_K2  ; Z
OUT VST80_K2_UPROG_1
LD TR0
AND C07_IND_VST80_K2  ; Z
OUT VST80_K2_UPROG_2
LD TR0
LD C08_IND_VST80_K2  ; Z
ANDNOT P_On
OR C79_IND_VST80_K2  ; Z
ANDLD
OUT VST80_K2_UPROG_3
LD TR0
LD 1206.00  ; C101_IND_VST80_K2
OR 1206.01  ; C102_IND_VST80_K2
OR 1206.02  ; C103_IND_VST80_K2
OR 1206.03  ; C104_IND_VST80_K2
ANDLD
OUT VST80_K2_UPROG_4
LD TR0
AND C50_IND_VST80_K2  ; Z
OUT VST80_K2_UPROG_5
LD TR0
AND C53_IND_VST80_K2  ; Z
OUT VST80_K2_UPROG_6
LD TR0
AND C52_IND_VST80_K2  ; Z
OUT VST80_K2_UPROG_7
LD TR0
LD C03_IND_VST80_K2  ; Z
OR C86_IND_VST80_K2  ; Z
OR C05_IND_VST80_K2  ; Z
OR C32_IND_VST80_K2  ; Z
ANDLD
OUT VST80_K2_UPROG_8
LD TR0
LD C83_IND_VST80_K2  ; Z
OR C84_IND_VST80_K2  ; Z
ANDLD
OUT VST80_K2_UPROG_9
LD TR0
LD C77_IND_VST80_K2  ; Z
OR C78_IND_VST80_K2  ; Z
ANDLD
OUT VST80_K2_UPROG_10
LD TR0
AND C54_IND_VST80_K2  ; Z
OUT VST80_K2_UPROG_11

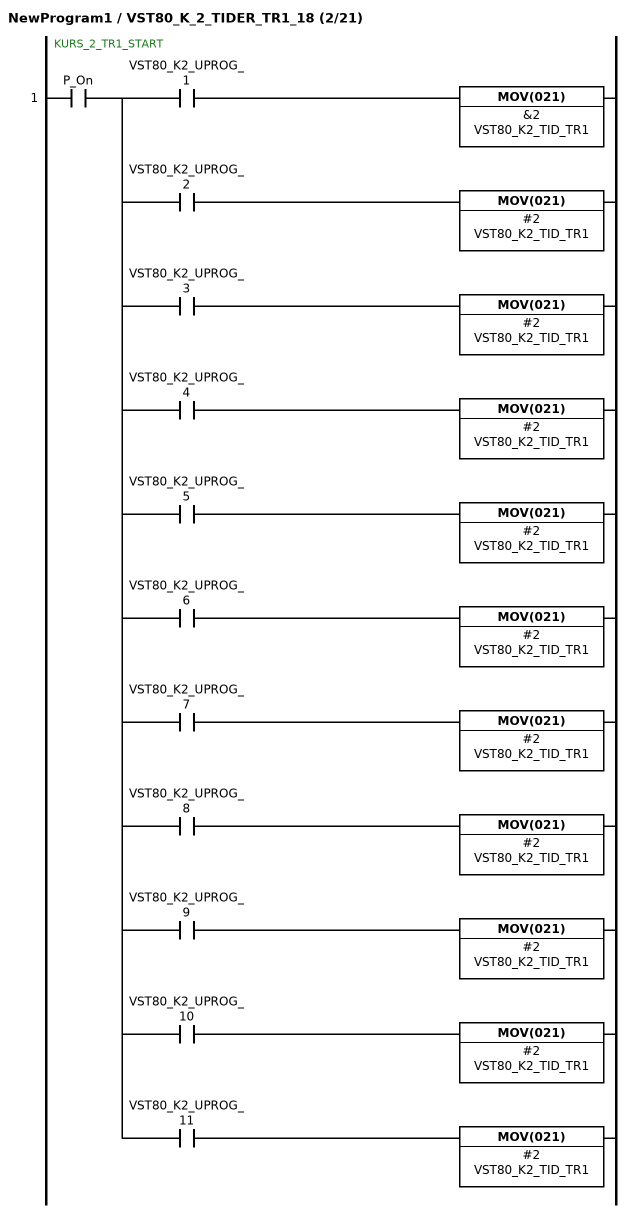
; rung 1: KURS_2_TR1_START
LD P_On
OUT TR0
AND VST80_K2_UPROG_1
MOV(021) &2 VST80_K2_TID_TR1
LD TR0
AND VST80_K2_UPROG_2
MOV(021) #2 VST80_K2_TID_TR1
LD TR0
AND VST80_K2_UPROG_3
MOV(021) #2 VST80_K2_TID_TR1
LD TR0
AND VST80_K2_UPROG_4
MOV(021) #2 VST80_K2_TID_TR1
LD TR0
AND VST80_K2_UPROG_5
MOV(021) #2 VST80_K2_TID_TR1
LD TR0
AND VST80_K2_UPROG_6
MOV(021) #2 VST80_K2_TID_TR1
LD TR0
AND VST80_K2_UPROG_7
MOV(021) #2 VST80_K2_TID_TR1
LD TR0
AND VST80_K2_UPROG_8
MOV(021) #2 VST80_K2_TID_TR1
LD TR0
AND VST80_K2_UPROG_9
MOV(021) #2 VST80_K2_TID_TR1
LD TR0
AND VST80_K2_UPROG_10
MOV(021) #2 VST80_K2_TID_TR1
LD TR0
AND VST80_K2_UPROG_11
MOV(021) #2 VST80_K2_TID_TR1

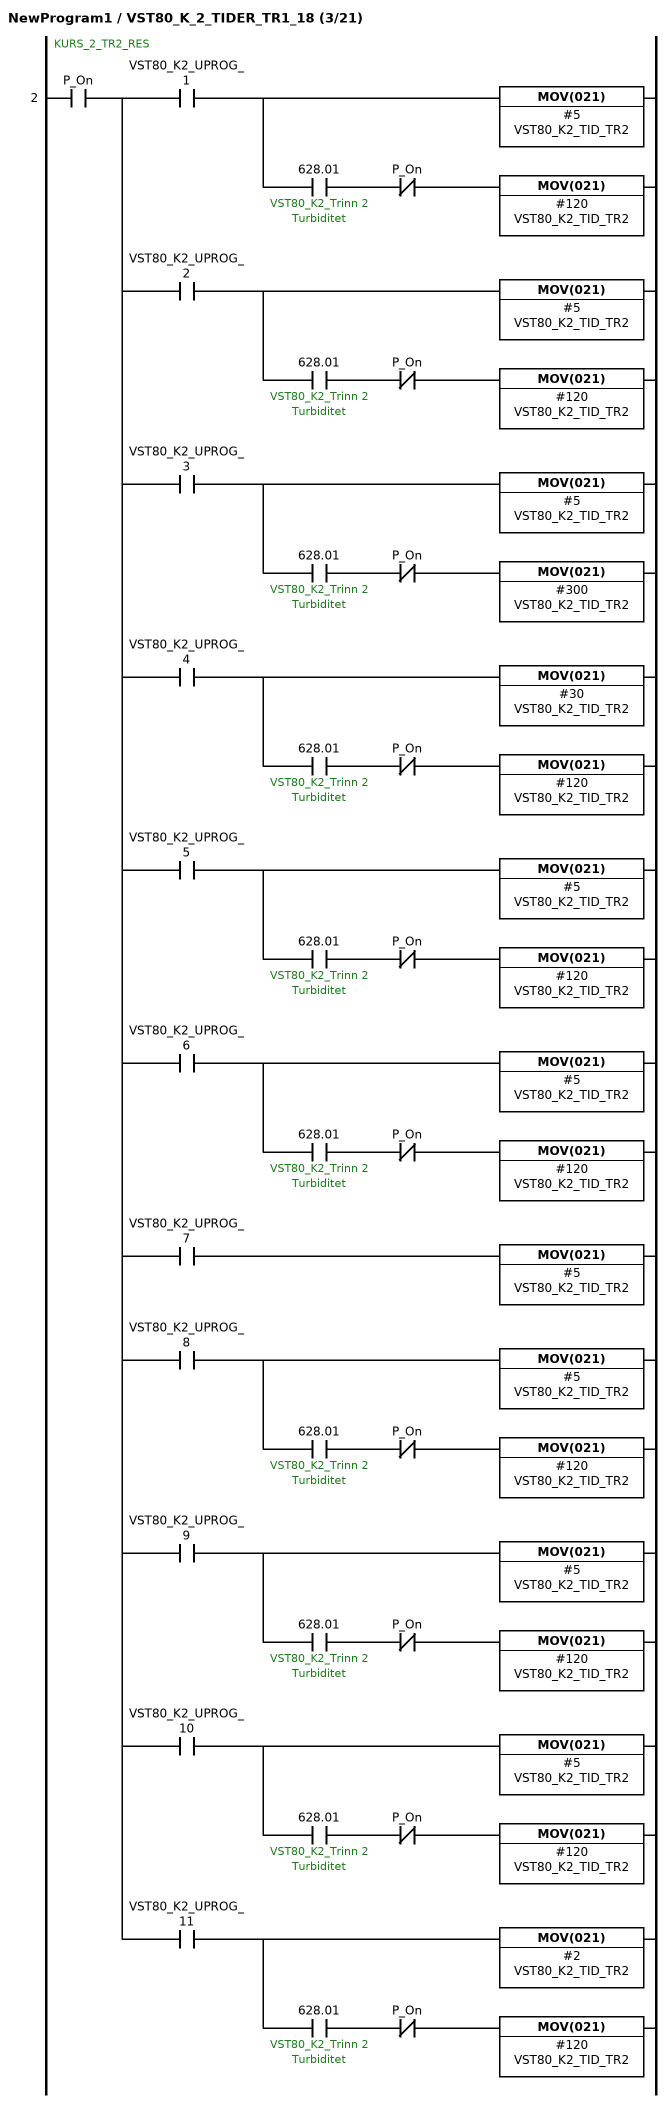
; rung 2: KURS_2_TR2_RES
LD P_On
OUT TR0
AND VST80_K2_UPROG_1
MOV(021) #5 VST80_K2_TID_TR2
AND 628.01  ; VST80_K2_Trinn 2 Turbiditet
ANDNOT P_On
MOV(021) #120 VST80_K2_TID_TR2
LD TR0
AND VST80_K2_UPROG_2
MOV(021) #5 VST80_K2_TID_TR2
AND 628.01  ; VST80_K2_Trinn 2 Turbiditet
ANDNOT P_On
MOV(021) #120 VST80_K2_TID_TR2
LD TR0
AND VST80_K2_UPROG_3
MOV(021) #5 VST80_K2_TID_TR2
AND 628.01  ; VST80_K2_Trinn 2 Turbiditet
ANDNOT P_On
MOV(021) #300 VST80_K2_TID_TR2
LD TR0
AND VST80_K2_UPROG_4
MOV(021) #30 VST80_K2_TID_TR2
AND 628.01  ; VST80_K2_Trinn 2 Turbiditet
ANDNOT P_On
MOV(021) #120 VST80_K2_TID_TR2
LD TR0
AND VST80_K2_UPROG_5
MOV(021) #5 VST80_K2_TID_TR2
AND 628.01  ; VST80_K2_Trinn 2 Turbiditet
ANDNOT P_On
MOV(021) #120 VST80_K2_TID_TR2
LD TR0
AND VST80_K2_UPROG_6
MOV(021) #5 VST80_K2_TID_TR2
AND 628.01  ; VST80_K2_Trinn 2 Turbiditet
ANDNOT P_On
MOV(021) #120 VST80_K2_TID_TR2
LD TR0
AND VST80_K2_UPROG_7
MOV(021) #5 VST80_K2_TID_TR2
LD TR0
AND VST80_K2_UPROG_8
MOV(021) #5 VST80_K2_TID_TR2
AND 628.01  ; VST80_K2_Trinn 2 Turbiditet
ANDNOT P_On
MOV(021) #120 VST80_K2_TID_TR2
LD TR0
AND VST80_K2_UPROG_9
MOV(021) #5 VST80_K2_TID_TR2
AND 628.01  ; VST80_K2_Trinn 2 Turbiditet
ANDNOT P_On
MOV(021) #120 VST80_K2_TID_TR2
LD TR0
AND VST80_K2_UPROG_10
MOV(021) #5 VST80_K2_TID_TR2
AND 628.01  ; VST80_K2_Trinn 2 Turbiditet
ANDNOT P_On
MOV(021) #120 VST80_K2_TID_TR2
LD TR0
AND VST80_K2_UPROG_11
MOV(021) #2 VST80_K2_TID_TR2
AND 628.01  ; VST80_K2_Trinn 2 Turbiditet
ANDNOT P_On
MOV(021) #120 VST80_K2_TID_TR2

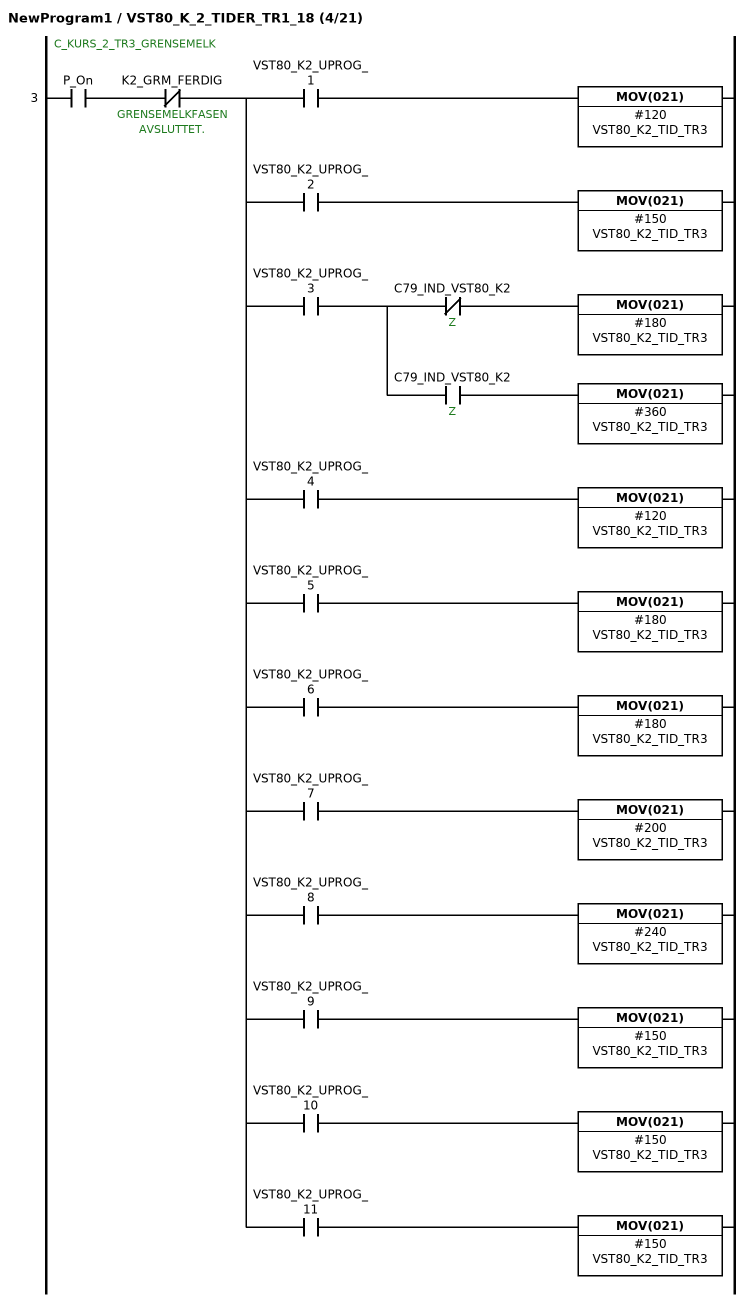
; rung 3: C_KURS_2_TR3_GRENSEMELK
LD P_On
ANDNOT K2_GRM_FERDIG  ; GRENSEMELKFASEN AVSLUTTET.
OUT TR0
AND VST80_K2_UPROG_1
MOV(021) #120 VST80_K2_TID_TR3
LD TR0
AND VST80_K2_UPROG_2
MOV(021) #150 VST80_K2_TID_TR3
LD TR0
AND VST80_K2_UPROG_3
OUT TR1
ANDNOT C79_IND_VST80_K2  ; Z
MOV(021) #180 VST80_K2_TID_TR3
LD TR1
AND C79_IND_VST80_K2  ; Z
MOV(021) #360 VST80_K2_TID_TR3
LD TR0
AND VST80_K2_UPROG_4
MOV(021) #120 VST80_K2_TID_TR3
LD TR0
AND VST80_K2_UPROG_5
MOV(021) #180 VST80_K2_TID_TR3
LD TR0
AND VST80_K2_UPROG_6
MOV(021) #180 VST80_K2_TID_TR3
LD TR0
AND VST80_K2_UPROG_7
MOV(021) #200 VST80_K2_TID_TR3
LD TR0
AND VST80_K2_UPROG_8
MOV(021) #240 VST80_K2_TID_TR3
LD TR0
AND VST80_K2_UPROG_9
MOV(021) #150 VST80_K2_TID_TR3
LD TR0
AND VST80_K2_UPROG_10
MOV(021) #150 VST80_K2_TID_TR3
LD TR0
AND VST80_K2_UPROG_11
MOV(021) #150 VST80_K2_TID_TR3

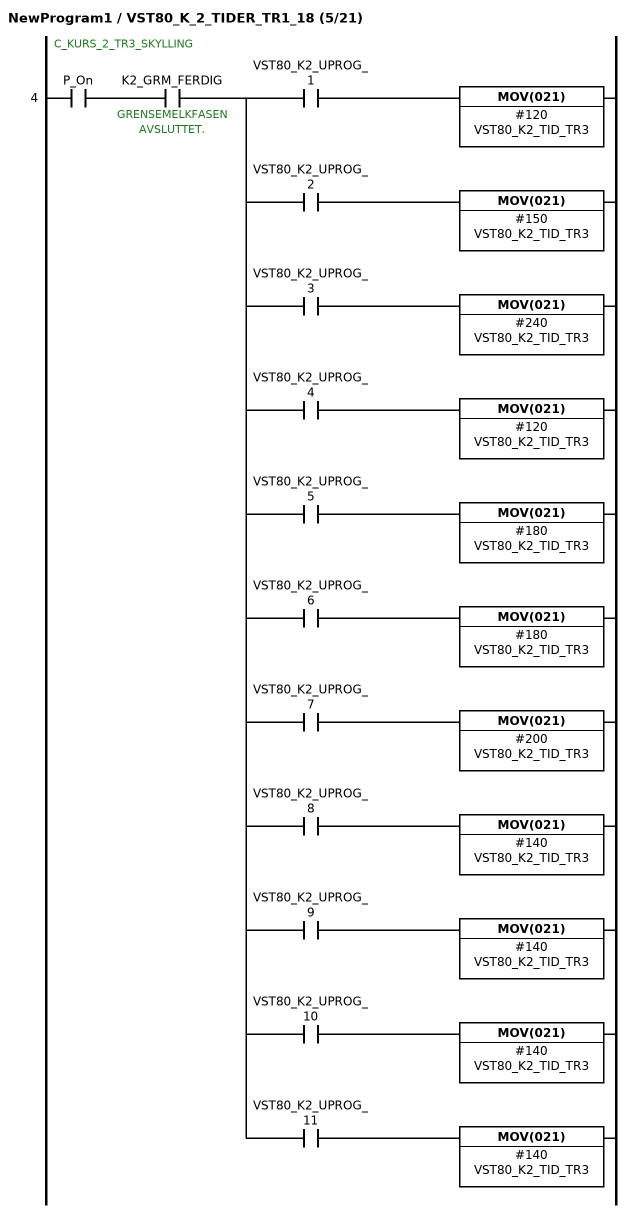
; rung 4: C_KURS_2_TR3_SKYLLING
LD P_On
AND K2_GRM_FERDIG  ; GRENSEMELKFASEN AVSLUTTET.
OUT TR0
AND VST80_K2_UPROG_1
MOV(021) #120 VST80_K2_TID_TR3
LD TR0
AND VST80_K2_UPROG_2
MOV(021) #150 VST80_K2_TID_TR3
LD TR0
AND VST80_K2_UPROG_3
MOV(021) #240 VST80_K2_TID_TR3
LD TR0
AND VST80_K2_UPROG_4
MOV(021) #120 VST80_K2_TID_TR3
LD TR0
AND VST80_K2_UPROG_5
MOV(021) #180 VST80_K2_TID_TR3
LD TR0
AND VST80_K2_UPROG_6
MOV(021) #180 VST80_K2_TID_TR3
LD TR0
AND VST80_K2_UPROG_7
MOV(021) #200 VST80_K2_TID_TR3
LD TR0
AND VST80_K2_UPROG_8
MOV(021) #140 VST80_K2_TID_TR3
LD TR0
AND VST80_K2_UPROG_9
MOV(021) #140 VST80_K2_TID_TR3
LD TR0
AND VST80_K2_UPROG_10
MOV(021) #140 VST80_K2_TID_TR3
LD TR0
AND VST80_K2_UPROG_11
MOV(021) #140 VST80_K2_TID_TR3

